(* CoDeSys 2.3.9.35 project: Q4_SISTEMA_DE_ESTEIRA.pro *)
(* Author: Franklin *)
(* Libraries: SysLibTargetVisu.lib 26.11.08 09:50:36, Standard.lib 26.11.08 09:46:20, Iecsfc.lib 26.11.08 09:46:14, DU35x.lib 26.11.09 14:36:14, SYSLIBCALLBACK.LIB 26.11.08 09:50:38 *)

(* PLC configuration (modules and I/O channels)
PLC Configuration [Root] node -1, in %IB0 out %QB0
  Communication [Comunica] node 0, in %IB0 out %QB0
    COM1 [COM1] node 0, in %IB0 out %QB0 {BaudRate = 115200; Paridade = No Parity; StopBits = 1 Stop Bit; Modem = Without RTS/CTS; Delay = 5}
      MToolIEC [Codesys] node 0, in %IB0 out %QB0
    COM2 [COM2] node 1, in %IB0 out %QB0 {BaudRate = 115200; Paridade = No Parity; StopBits = 1 Stop Bit; Modem = Without RTS/CTS; Delay = 5}
      Disable [Desabilitado485] node 0, in %IB0 out %QB0
  Bus [Barramento] node 1, in %IB0 out %QB0
    Inputs [Entradas] node 0, in %IB0 out %QB0
      Digital Inputs 0 [Entradas0] node 0, in %IW0 out %QB0
        I00 AT %IX0.0 [BitInput] I0.0
        I01 AT %IX0.1 [BitInput] I0.1
        I02 AT %IX0.2 [BitInput] I0.2
        I03 AT %IX0.3 [BitInput] I0.3
        I04 AT %IX0.4 [BitInput] I0.4
        I05 AT %IX0.5 [BitInput] I0.5
        I06 AT %IX0.6 [BitInput] I0.6
        I07 AT %IX0.7 [BitInput] I0.7
        I08 AT %IX0.8 [BitInput] I0.8
      Digital Inputs 1 [Entradas1] node 0, in %IW1 out %QB0
        I10 AT %IX1.0 [BitInput] I1.0
        I11 AT %IX1.1 [BitInput] I1.1
        I12 AT %IX1.2 [BitInput] I1.2
        I13 AT %IX1.3 [BitInput] I1.3
        I14 AT %IX1.4 [BitInput] I1.4
        I15 AT %IX1.5 [BitInput] I1.5
        I16 AT %IX1.6 [BitInput] I1.6
        I17 AT %IX1.7 [BitInput] I1.7
        I18 AT %IX1.8 [BitInput] I1.8
      Digital Inputs 2 [Entradas2] node 0, in %IW2 out %QB0
        I20 AT %IX2.0 [BitInput] I2.0
        I21 AT %IX2.1 [BitInput] I2.1
      Analog Inputs [EntradaAnalogica] node 0, in %IW4 out %QB0
        AI0 AT %IW4 [WordInput] AI0 {TipoAnalogica = Channel Disable; FiltroAnalogica = Filter 0 - AI=2ms  / AV=90ms; FundoEscala = 0}
        AI1 AT %IW5 [WordInput] AI1 {TipoAnalogica = Channel Disable; FiltroAnalogica = Filter 0 - AI=2ms  / AV=90ms; FundoEscala = 0}
        AI2 AT %IW6 [WordInput] AI2 {TipoAnalogica = Channel Disable; FiltroAnalogica = Filter 0 - AI=2ms  / AV=90ms; FundoEscala = 0}
        AI3 AT %IW7 [WordInput] AI3 {TipoAnalogica = Channel Disable; FiltroAnalogica = Filter 0 - AI=2ms  / AV=90ms; FundoEscala = 0}
      Fast Inputs [EntradasRapidas] node 1, in %IB16 out %QB0
        Block 0 [Bloco0] node 0, in %IB16 out %QB0
          Disable [DesabilitadoBloco0] node 0, in %IB16 out %QB0
        Block 1 [Bloco1] node 1, in %IB16 out %QB0
          Disable [DesabilitadoBloco1] node 0, in %IB16 out %QB0
        Configurable Input Block 0 [EntradaConfiBloco0] node 2, in %IB16 out %QB0
          Counter 0 [EntradaConfContador0] node 0, in %IB16 out %QB0 {EntradaConfiguravelContador = Disable}
        Configurable Input Block 1 [EntradaConfiBloco1] node 3, in %IB16 out %QB0
          Counter 2 [EntradaConfContador2] node 0, in %IB16 out %QB0 {EntradaConfiguravelContador = Disable}
    Outputs [Saidas] node 1, in %IB13 out %QB0
      Digital Outputs 0 [Saidas0] node 0, in %IW0 out %QW0
        Q00 AT %QX0.0 [BitOutput] Q0.0
        Q01 AT %QX0.1 [BitOutput] Q0.1
        Q02 AT %QX0.2 [BitOutput] Q0.2
        Q03 AT %QX0.3 [BitOutput] Q0.3
        Q04 AT %QX0.4 [BitOutput] Q0.4
        Q05 AT %QX0.5 [BitOutput] Q0.5
        Q06 AT %QX0.6 [BitOutput] Q0.6
        Q07 AT %QX0.7 [BitOutput] Q0.7
      Digital Outputs 1 [Saidas1] node 0, in %IW0 out %QW1
        Q10 AT %QX1.0 [BitOutput] Q1.0
        Q11 AT %QX1.1 [BitOutput] Q1.1
        Q12 AT %QX1.2 [BitOutput] Q1.2
        Q13 AT %QX1.3 [BitOutput] Q1.3
        Q14 AT %QX1.4 [BitOutput] Q1.4
        Q15 AT %QX1.5 [BitOutput] Q1.5
        Q16 AT %QX1.6 [BitOutput] Q1.6
        Q17 AT %QX1.7 [BitOutput] Q1.7
      Analog Outputs [SaidaAnalogica] node 0, in %IW0 out %QW3
        AO0 AT %QW3 [WordOutput] AO0 {TipoAnalogica = Channel Disable; FundoEscala = 0}
        AO1 AT %QW4 [WordOutput] AO1 {TipoAnalogica = Channel Disable; FundoEscala = 0}
      Fast Outputs [SaidasRapidas] node 1, in %IB0 out %QB10
        Fast Output 0 Disable [DesabilitadoF0] node 0, in %IB0 out %QB10
        Fast Output 1 Disable [DesabilitadoF1] node 1, in %IB0 out %QB10
      Counter Output [SaidasContador] node 2, in %IB0 out %QB10
        Block 0 Output Disable [DesabilitadoSaidaBloco0] node 0, in %IB0 out %QB10
        Block 1 Output Disable [DesabilitadoSaidaBloco1] node 1, in %IB0 out %QB10
  External Events [Eventos] node 2, in %IB13 out %QB6
    Timer Event [TimerEvent] node 0, in %IB13 out %QB6 {Intervalo = 10}
*)

(* POU PLC_PRG, LD *)
PROGRAM PLC_PRG
VAR
	S0 AT %MX1.0: BOOL;
	CH AT %IX0.1: BOOL;
	SP AT %IX0.0: BOOL;
	QCU AT %MX0.1: BOOL;
	T0 AT %MX2.0: BOOL;
	S1 AT %MX1.1: BOOL;
	T1 AT %MX2.1: BOOL;
	S2 AT %MX1.2: BOOL;
	T2 AT %MX2.2: BOOL;
	S3 AT %MX1.3: BOOL;
	QT1 AT %MX0.3: BOOL;
	T3 AT %MX2.3: BOOL;
	S4 AT %MX1.4: BOOL;
	T4 AT %MX2.4: BOOL;
	CA AT %QX0.0: BOOL;
	CB AT %QX0.1: BOOL;
	CC AT %QX0.2: BOOL;
	M AT %QX0.3: BOOL;
	CU AT %MX0.0: BOOL;
	P: R_TRIG;
	T1_EN AT %MX0.2: BOOL;
	TEMPORIZADOR1: TON;
	CTU: CTU;
	COUNT AT %MW10: INT;
END_VAR
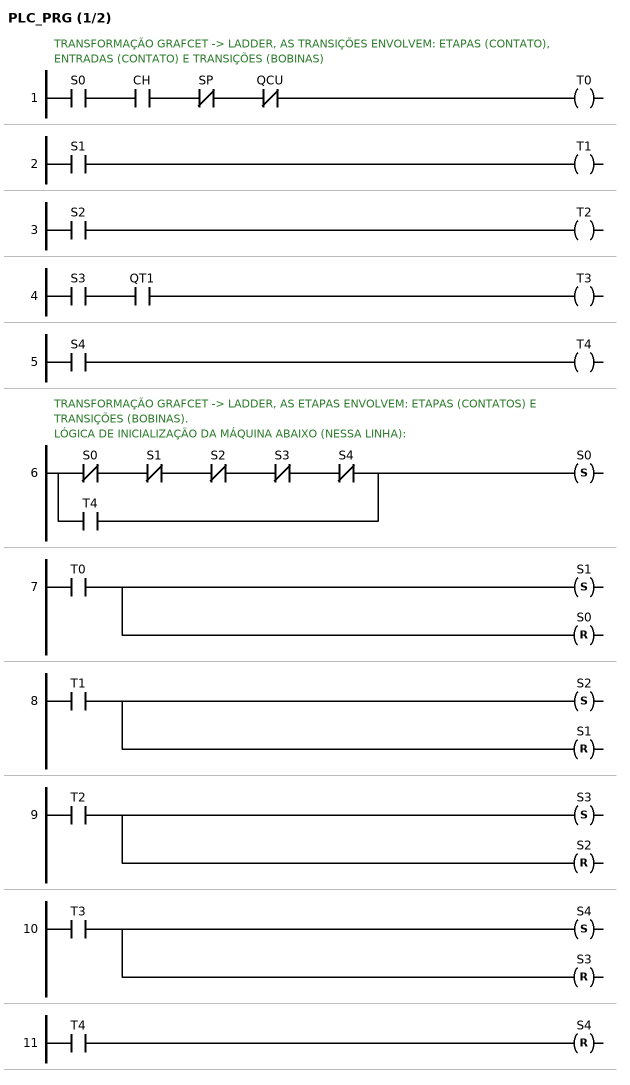
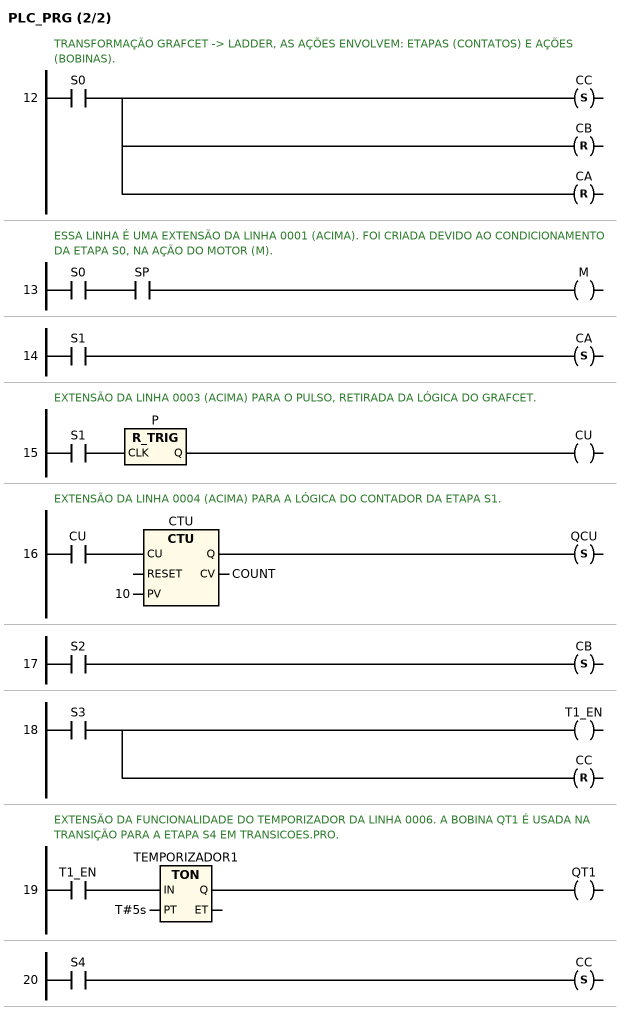
_LD_ (* Ladder Diagram *)
NETWORK 1 (* TRANSFORMAÇÃO GRAFCET -> LADDER, AS TRANSIÇÕES ENVOLVEM: ETAPAS (CONTATO), ENTRADAS (CONTATO) E TRANSIÇÕES (BOBINAS) *)
	[S0] - [CH] - [/SP] - [/QCU] --- (T0)
NETWORK 2
	[S1] --- (T1)
NETWORK 3
	[S2] --- (T2)
NETWORK 4
	[S3] - [QT1] --- (T3)
NETWORK 5
	[S4] --- (T4)
NETWORK 6 (* TRANSFORMAÇÃO GRAFCET -> LADDER, AS ETAPAS ENVOLVEM: ETAPAS (CONTATOS) E TRANSIÇÕES (BOBINAS). / LÓGICA DE INICIALIZAÇÃO DA MÁQUINA ABAIXO (NESSA LINHA): *)
	{ [/S0] - [/S1] - [/S2] - [/S3] - [/S4] | [T4] } --- (S S0)
NETWORK 7
	[T0] --- (S S1) (R S0)
NETWORK 8
	[T1] --- (S S2) (R S1)
NETWORK 9
	[T2] --- (S S3) (R S2)
NETWORK 10
	[T3] --- (S S4) (R S3)
NETWORK 11
	[T4] --- (R S4)
NETWORK 12 (* TRANSFORMAÇÃO GRAFCET -> LADDER, AS AÇÕES ENVOLVEM: ETAPAS (CONTATOS) E AÇÕES (BOBINAS). *)
	[S0] --- (S CC) (R CB) (R CA)
NETWORK 13 (* ESSA LINHA É UMA EXTENSÃO DA LINHA 0001 (ACIMA). FOI CRIADA DEVIDO AO CONDICIONAMENTO DA ETAPA S0, NA AÇÃO DO MOTOR (M). *)
	[S0] - [SP] --- (M)
NETWORK 14
	[S1] --- (S CA)
NETWORK 15 (* EXTENSÃO DA LINHA 0003 (ACIMA) PARA O PULSO, RETIRADA DA LÓGICA DO GRAFCET. *)
	[S1] - P:R_TRIG(CLK: *) --- (CU)
NETWORK 16 (* EXTENSÃO DA LINHA 0004 (ACIMA) PARA A LÓGICA DO CONTADOR DA ETAPA S1. *)
	[CU] - CTU:CTU(CU: *, RESET: , PV: 10, CV => COUNT) --- (S QCU)
NETWORK 17
	[S2] --- (S CB)
NETWORK 18
	[S3] --- (T1_EN) (R CC)
NETWORK 19 (* EXTENSÃO DA FUNCIONALIDADE DO TEMPORIZADOR DA LINHA 0006. A BOBINA QT1 É USADA NA TRANSIÇÃO PARA A ETAPA S4 EM TRANSICOES.PRO. *)
	[T1_EN] - TEMPORIZADOR1:TON(IN: *, PT: T#5s) --- (QT1)
NETWORK 20
	[S4] --- (S CC)
_END_LD_
(* the same logic as Structured Text *)
(* Network 1 *)
T0 := S0 AND CH AND NOT SP AND NOT QCU;
(* Network 2 *)
T1 := S1;
(* Network 3 *)
T2 := S2;
(* Network 4 *)
T3 := S3 AND QT1;
(* Network 5 *)
T4 := S4;
(* Network 6 *)
IF NOT S0 AND NOT S1 AND NOT S2 AND NOT S3 AND NOT S4 OR T4 THEN S0 := TRUE; END_IF;
(* Network 7 *)
IF T0 THEN S1 := TRUE; S0 := FALSE; END_IF;
(* Network 8 *)
IF T1 THEN S2 := TRUE; S1 := FALSE; END_IF;
(* Network 9 *)
IF T2 THEN S3 := TRUE; S2 := FALSE; END_IF;
(* Network 10 *)
IF T3 THEN S4 := TRUE; S3 := FALSE; END_IF;
(* Network 11 *)
IF T4 THEN S4 := FALSE; END_IF;
(* Network 12 *)
IF S0 THEN CC := TRUE; CB := FALSE; CA := FALSE; END_IF;
(* Network 13 *)
M := S0 AND SP;
(* Network 14 *)
IF S1 THEN CA := TRUE; END_IF;
(* Network 15 *)
P(CLK := S1);
CU := P.Q;
(* Network 16: see the listing above *)
(* Network 17 *)
IF S2 THEN CB := TRUE; END_IF;
(* Network 18 *)
T1_EN := S3;
IF S3 THEN CC := FALSE; END_IF;
(* Network 19 *)
TEMPORIZADOR1(IN := T1_EN, PT := T#5s);
QT1 := TEMPORIZADOR1.Q;
(* Network 20 *)
IF S4 THEN CC := TRUE; END_IF;
END_PROGRAM
ACTION ACOES:
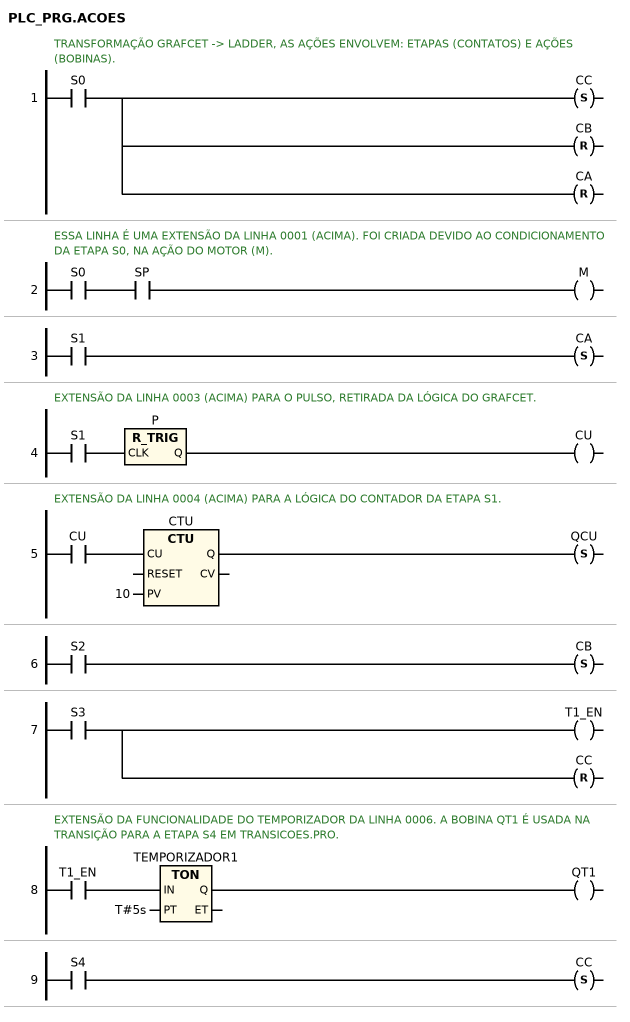
_LD_ (* Ladder Diagram *)
NETWORK 1 (* TRANSFORMAÇÃO GRAFCET -> LADDER, AS AÇÕES ENVOLVEM: ETAPAS (CONTATOS) E AÇÕES (BOBINAS). *)
	[S0] --- (S CC) (R CB) (R CA)
NETWORK 2 (* ESSA LINHA É UMA EXTENSÃO DA LINHA 0001 (ACIMA). FOI CRIADA DEVIDO AO CONDICIONAMENTO DA ETAPA S0, NA AÇÃO DO MOTOR (M). *)
	[S0] - [SP] --- (M)
NETWORK 3
	[S1] --- (S CA)
NETWORK 4 (* EXTENSÃO DA LINHA 0003 (ACIMA) PARA O PULSO, RETIRADA DA LÓGICA DO GRAFCET. *)
	[S1] - P:R_TRIG(CLK: *) --- (CU)
NETWORK 5 (* EXTENSÃO DA LINHA 0004 (ACIMA) PARA A LÓGICA DO CONTADOR DA ETAPA S1. *)
	[CU] - CTU:CTU(CU: *, RESET: , PV: 10) --- (S QCU)
NETWORK 6
	[S2] --- (S CB)
NETWORK 7
	[S3] --- (T1_EN) (R CC)
NETWORK 8 (* EXTENSÃO DA FUNCIONALIDADE DO TEMPORIZADOR DA LINHA 0006. A BOBINA QT1 É USADA NA TRANSIÇÃO PARA A ETAPA S4 EM TRANSICOES.PRO. *)
	[T1_EN] - TEMPORIZADOR1:TON(IN: *, PT: T#5s) --- (QT1)
NETWORK 9
	[S4] --- (S CC)
_END_LD_
(* the same logic as Structured Text *)
(* Network 1 *)
IF S0 THEN CC := TRUE; CB := FALSE; CA := FALSE; END_IF;
(* Network 2 *)
M := S0 AND SP;
(* Network 3 *)
IF S1 THEN CA := TRUE; END_IF;
(* Network 4 *)
P(CLK := S1);
CU := P.Q;
(* Network 5: see the listing above *)
(* Network 6 *)
IF S2 THEN CB := TRUE; END_IF;
(* Network 7 *)
T1_EN := S3;
IF S3 THEN CC := FALSE; END_IF;
(* Network 8 *)
TEMPORIZADOR1(IN := T1_EN, PT := T#5s);
QT1 := TEMPORIZADOR1.Q;
(* Network 9 *)
IF S4 THEN CC := TRUE; END_IF;
END_ACTION
ACTION ETAPAS:
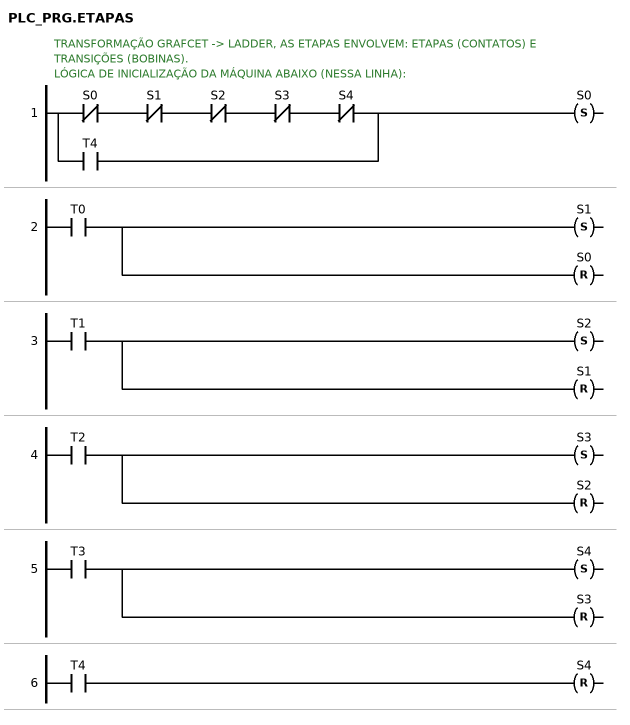
_LD_ (* Ladder Diagram *)
NETWORK 1 (* TRANSFORMAÇÃO GRAFCET -> LADDER, AS ETAPAS ENVOLVEM: ETAPAS (CONTATOS) E TRANSIÇÕES (BOBINAS). / LÓGICA DE INICIALIZAÇÃO DA MÁQUINA ABAIXO (NESSA LINHA): *)
	{ [/S0] - [/S1] - [/S2] - [/S3] - [/S4] | [T4] } --- (S S0)
NETWORK 2
	[T0] --- (S S1) (R S0)
NETWORK 3
	[T1] --- (S S2) (R S1)
NETWORK 4
	[T2] --- (S S3) (R S2)
NETWORK 5
	[T3] --- (S S4) (R S3)
NETWORK 6
	[T4] --- (R S4)
_END_LD_
(* the same logic as Structured Text *)
(* Network 1: TRANSFORMAÇÃO GRAFCET -> LADDER, AS ETAPAS ENVOLVEM: ETAPAS (CONTATOS) E TRANSIÇÕES (BOBINAS). / LÓGICA DE INICIALIZAÇÃO DA MÁQUINA ABAIXO (NESSA LINHA): *)
IF NOT S0 AND NOT S1 AND NOT S2 AND NOT S3 AND NOT S4 OR T4 THEN S0 := TRUE; END_IF;
(* Network 2 *)
IF T0 THEN S1 := TRUE; S0 := FALSE; END_IF;
(* Network 3 *)
IF T1 THEN S2 := TRUE; S1 := FALSE; END_IF;
(* Network 4 *)
IF T2 THEN S3 := TRUE; S2 := FALSE; END_IF;
(* Network 5 *)
IF T3 THEN S4 := TRUE; S3 := FALSE; END_IF;
(* Network 6 *)
IF T4 THEN S4 := FALSE; END_IF;
END_ACTION
ACTION TRANSICOES:
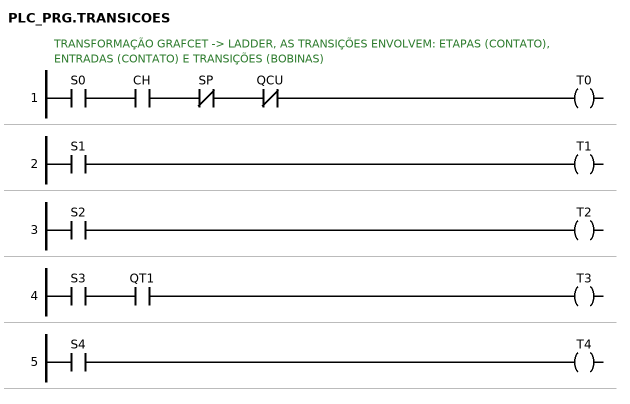
_LD_ (* Ladder Diagram *)
NETWORK 1 (* TRANSFORMAÇÃO GRAFCET -> LADDER, AS TRANSIÇÕES ENVOLVEM: ETAPAS (CONTATO), ENTRADAS (CONTATO) E TRANSIÇÕES (BOBINAS) *)
	[S0] - [CH] - [/SP] - [/QCU] --- (T0)
NETWORK 2
	[S1] --- (T1)
NETWORK 3
	[S2] --- (T2)
NETWORK 4
	[S3] - [QT1] --- (T3)
NETWORK 5
	[S4] --- (T4)
_END_LD_
(* the same logic as Structured Text *)
(* Network 1: TRANSFORMAÇÃO GRAFCET -> LADDER, AS TRANSIÇÕES ENVOLVEM: ETAPAS (CONTATO), ENTRADAS (CONTATO) E TRANSIÇÕES (BOBINAS) *)
T0 := S0 AND CH AND NOT SP AND NOT QCU;
(* Network 2 *)
T1 := S1;
(* Network 3 *)
T2 := S2;
(* Network 4 *)
T3 := S3 AND QT1;
(* Network 5 *)
T4 := S4;
END_ACTION

(* Visualisation v1
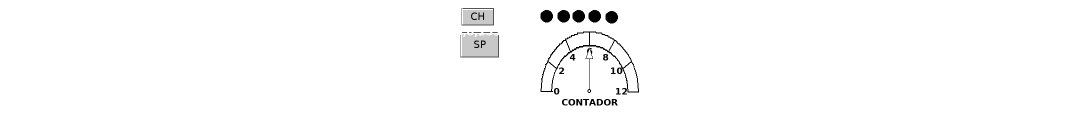
button at (4,3)-(36,20): text "CH"; toggles PLC_PRG.CH
button at (3,27)-(41,52): text "SP"; toggles PLC_PRG.SP
ellipse at (83,5)-(95,17): text "S0"; alarm colour if PLC_PRG.S0
ellipse at (100,5)-(112,17): text "S1"; alarm colour if PLC_PRG.S1
ellipse at (115,5)-(127,17): text "S2"; alarm colour if PLC_PRG.S2
ellipse at (131,5)-(143,17): text "S3"; alarm colour if PLC_PRG.S3
ellipse at (148,6)-(160,18): text "S4"; alarm colour if PLC_PRG.S4
group at (82,26)-(181,106)
  rectangle at (0,0)-(1,1): text "{ExtendedElement},Visu\ElementDLL.ete,0,@Zeigerinstrument,99,180,0,0,255,255,255,0,PLC_PRG.COUNT,CONTADOR,%.0f,1,1,1,2,2,0,12,0,0,0,0,0,0,0,-11,80,700,Arial,1,0,"
  rectangle at (14,43)-(20,57): text "0"
  rectangle at (19,26)-(25,40): text "2"
  rectangle at (30,15)-(36,29): text "4"
  rectangle at (47,10)-(53,24): text "6"
  rectangle at (63,15)-(69,29): text "8"
  rectangle at (71,26)-(83,40): text "10"
  rectangle at (76,43)-(88,57): text "12"
  rectangle at (20,52)-(80,66): text "CONTADOR"
  polygon at (46,14)-(53,50): angle ((PLC_PRG.COUNT * 1.0)-6) * 15
10 more shapes without text or variables
*)
